// Example 1 - ConstantGap: ONE cam table, 9 points.
//
//   Mover 1 = master, runs at constant velocity around the track.
//   Mover 2 = slave, follows Mover 1 through a cam table that covers one full lap (1500 mm).
//
// Mover 2 is 100 mm behind Mover 1 on the straights and 60 mm in the curves, blended over TRANSITION mm
// at the start of every section. The table is written by hand in the action BuildTable (F_CamPoint).
//
// How to run (online view, with MAIN.eExample = ConstantGap):  bStart -> watch eState -> bStop.   On Error: bReset.
// Watch fGapActual while it runs: 100 on the straights, 60 in the curves, a smooth blend at each section start.
PROGRAM PRG_Example1
VAR CONSTANT
	// --- track geometry (mm) ---
	TRACK_LENGTH			: LREAL := 1500.0;	// = modulo factor of both mover axes
	STRAIGHT_1_START		: LREAL := 0.0;
	CURVE_1_START			: LREAL := 250.0;
	STRAIGHT_2_START		: LREAL := 750.0;
	CURVE_2_START			: LREAL := 1000.0;

	// --- wanted distance Mover 1 -> Mover 2 (mm, Mover 2 runs BEHIND Mover 1) ---
	GAP_STRAIGHT			: LREAL := 100.0;
	GAP_CURVE				: LREAL := 60.0;
	TRANSITION				: LREAL := 100.0;	// master travel over which the gap blends to the new value

	// --- demo dynamics ---
	MASTER_VELOCITY			: LREAL := 300.0;	// mm/s, Mover 1 while running
	POSITIONING_VELOCITY	: LREAL := 200.0;	// mm/s, Mover 2 while pre-positioning

	CAM_TABLE_ID			: MC_CAM_ID := 1;	// NC > Tables > Table 1 (Ex 1-4) > Mover 2
	CAM_POINTS				: UDINT := 9;
END_VAR
VAR
	// --- commands: set TRUE in the online view, they reset themselves ---
	bStart				: BOOL;
	bStop				: BOOL;
	bReset				: BOOL;
	eState				: E_State;

	// --- cam table data: CAM_POINTS points, loaded into NC table CAM_TABLE_ID ---
	aCamPoints			: ARRAY[1..CAM_POINTS] OF MC_MotionFunctionPoint;
	stCamTable			: MC_CAM_REF;

	// --- function blocks ---
	fbPowerMover1		: MC_Power;
	fbPowerMover2		: MC_Power;
	fbResetMover1		: MC_Reset;
	fbResetMover2		: MC_Reset;
	fbCamTableSelect	: MC_CamTableSelect;			// PLC array -> NC cam table
	fbReadTable			: MC_ReadCamTableSlaveDynamics;	// "where does the table want the slave for this master position?"
	fbMoveRelMover2		: MC_MoveRelative;
	fbCamIn				: MC_CamIn;
	fbMoveVeloMover1	: MC_MoveVelocity;
	fbHaltMover1		: MC_Halt;
	fbCamOut			: MC_CamOut;

	// --- live values worth watching ---
	fMover1Pos			: LREAL;	// modulo set position of Mover 1 (0..1500)
	fMover2Pos			: LREAL;	// modulo set position of Mover 2 (0..1500)
	fGapActual			: LREAL;	// how far Mover 2 is behind Mover 1 right now (along the track)
	fGapWanted			: LREAL;	// what the table asked for at coupling time
	bError				: BOOL;
	nErrorID			: UDINT;
END_VAR

// update axis status every cycle
GVL_Axes.Mover1();
GVL_Axes.Mover2();

// live gap: Mover 1 position minus Mover 2 position, wrapped to 0..1500
fMover1Pos := GVL_Axes.Mover1.NcToPlc.ModuloSetPos;
fMover2Pos := GVL_Axes.Mover2.NcToPlc.ModuloSetPos;
fGapActual := fMover1Pos - fMover2Pos;
IF fGapActual < 0.0 THEN
	fGapActual := fGapActual + TRACK_LENGTH;
END_IF

CASE eState OF
	E_State.Idle:
		IF bStart THEN
			bStart := FALSE;
			eState := E_State.Enable;
		END_IF

	E_State.Enable:
		fbPowerMover1.Enable := TRUE;
		fbPowerMover1.Enable_Positive := TRUE;
		fbPowerMover1.Enable_Negative := TRUE;
		fbPowerMover2.Enable := TRUE;
		fbPowerMover2.Enable_Positive := TRUE;
		fbPowerMover2.Enable_Negative := TRUE;
		IF fbPowerMover1.Status AND fbPowerMover2.Status THEN
			eState := E_State.Decouple;
		END_IF

	E_State.Decouple:
		// An earlier run may have left Mover 2 coupled: the NC keeps the coupling through an axis error and MC_Reset
		// does not clear it. MC_CamTableSelect refuses to overwrite a table that a coupled axis is using (0x4A26).
		IF NOT fbCamOut.Execute THEN
			IF GVL_Axes.Mover2.Status.Coupled THEN
				fbCamOut.Execute := TRUE;
			ELSE
				eState := E_State.BuildTable;
			END_IF
		ELSIF fbCamOut.Done THEN
			fbCamOut.Execute := FALSE;
			eState := E_State.BuildTable;
		END_IF

	E_State.BuildTable:
		// fill the point array once, then hand it to the NC (overwrites cam table CAM_TABLE_ID)
		IF NOT fbCamTableSelect.Execute THEN
			BuildTable();
		END_IF
		fbCamTableSelect.Periodic := TRUE;		// one table = one lap, repeat forever
		fbCamTableSelect.CamTableID := CAM_TABLE_ID;
		fbCamTableSelect.Execute := TRUE;
		IF fbCamTableSelect.Done THEN
			fbCamTableSelect.Execute := FALSE;
			eState := E_State.ReadTable;
		END_IF

	E_State.ReadTable:
		// Mover 1 stays where it is. Ask the NC what slave position the table wants for it.
		// The table master runs 0..1500 = the track, so Mover 1's track position goes in as it is.
		fbReadTable.CamTableID := CAM_TABLE_ID;
		fbReadTable.MasterPosition := fMover1Pos;
		fbReadTable.Execute := TRUE;
		IF fbReadTable.Done THEN
			fbReadTable.Execute := FALSE;
			// table: slave = master - gap   ->   gap = master - slave
			fGapWanted := fMover1Pos - fbReadTable.SlavePosition;
			// Mover 1 stands still, so this relative move can never run into it:
			// positive = Mover 2 closes up from behind, negative = Mover 2 backs off a little
			fbMoveRelMover2.Distance := fGapActual - fGapWanted;
			eState := E_State.Preposition;
		END_IF

	E_State.Preposition:
		fbMoveRelMover2.Velocity := POSITIONING_VELOCITY;
		fbMoveRelMover2.Execute := TRUE;
		IF fbMoveRelMover2.Done THEN
			fbMoveRelMover2.Execute := FALSE;
			eState := E_State.CamIn;
		END_IF

	E_State.CamIn:
		fbCamIn.CamTableID := CAM_TABLE_ID;
		fbCamIn.StartMode := MC_STARTMODE_ABSOLUTE;		// table master axis = Mover 1 track position
		fbCamIn.MasterOffset := 0.0;
		fbCamIn.SlaveOffset := 0.0;
		fbCamIn.MasterScaling := 1.0;
		fbCamIn.SlaveScaling := 1.0;
		// let the NC pick the slave offset so Mover 2 never jumps at coupling.
		// After the pre-positioning above that offset is 0 (or whole laps), so the table gaps apply 1:1.
		fbCamIn.Options.SlaveScalingMode := MC_CAMSCALING_AUTOOFFSET;
		fbCamIn.Execute := TRUE;
		IF fbCamIn.InSync THEN
			fbCamIn.Execute := FALSE;
			eState := E_State.Run;
		END_IF

	E_State.Run:
		// only the master is commanded - the slave is driven by the cam
		fbMoveVeloMover1.Velocity := MASTER_VELOCITY;
		fbMoveVeloMover1.Direction := MC_Positive_Direction;
		fbMoveVeloMover1.Execute := TRUE;
		IF bStop THEN
			bStop := FALSE;
			fbMoveVeloMover1.Execute := FALSE;
			eState := E_State.Stopping;
		END_IF

	E_State.Stopping:
		fbHaltMover1.Execute := TRUE;
		IF fbHaltMover1.Done THEN
			fbHaltMover1.Execute := FALSE;
			eState := E_State.CamOut;
		END_IF

	E_State.CamOut:
		fbCamOut.Execute := TRUE;
		IF fbCamOut.Done THEN
			fbCamOut.Execute := FALSE;
			eState := E_State.Idle;
		END_IF

	E_State.Error:
		fbCamTableSelect.Execute := FALSE;
		fbReadTable.Execute := FALSE;
		fbMoveRelMover2.Execute := FALSE;
		fbCamIn.Execute := FALSE;
		fbMoveVeloMover1.Execute := FALSE;
		// a slave error does not stop the master: halt Mover 1 if it is still running and not in error itself
		fbHaltMover1.Execute := NOT GVL_Axes.Mover1.Status.Error AND GVL_Axes.Mover1.Status.Moving;
		fbCamOut.Execute := FALSE;
		IF bReset THEN
			bReset := FALSE;
			fbResetMover1.Execute := TRUE;
			fbResetMover2.Execute := TRUE;
			eState := E_State.Resetting;
		END_IF

	E_State.Resetting:
		IF (fbResetMover1.Done OR fbResetMover1.Error) AND (fbResetMover2.Done OR fbResetMover2.Error) THEN
			fbResetMover1.Execute := FALSE;
			fbResetMover2.Execute := FALSE;
			bError := FALSE;
			nErrorID := 0;
			eState := E_State.Idle;
		END_IF
END_CASE

// any error anywhere -> Error state
IF eState <> E_State.Error AND eState <> E_State.Resetting THEN
	IF GVL_Axes.Mover1.Status.Error THEN
		nErrorID := GVL_Axes.Mover1.Status.ErrorID;
	ELSIF GVL_Axes.Mover2.Status.Error THEN
		nErrorID := GVL_Axes.Mover2.Status.ErrorID;
	ELSIF fbPowerMover1.Error THEN
		nErrorID := fbPowerMover1.ErrorID;
	ELSIF fbPowerMover2.Error THEN
		nErrorID := fbPowerMover2.ErrorID;
	ELSIF fbCamTableSelect.Error THEN
		nErrorID := fbCamTableSelect.ErrorID;
	ELSIF fbReadTable.Error THEN
		nErrorID := fbReadTable.ErrorID;
	ELSIF fbMoveRelMover2.Error THEN
		nErrorID := fbMoveRelMover2.ErrorID;
	ELSIF fbCamIn.Error THEN
		nErrorID := fbCamIn.ErrorID;
	ELSIF fbMoveVeloMover1.Error THEN
		nErrorID := fbMoveVeloMover1.ErrorID;
	ELSIF fbHaltMover1.Error THEN
		nErrorID := fbHaltMover1.ErrorID;
	ELSIF fbCamOut.Error THEN
		nErrorID := fbCamOut.ErrorID;
	END_IF
	IF nErrorID <> 0 THEN
		bError := TRUE;
		eState := E_State.Error;
	END_IF
END_IF

// call every function block once per cycle
fbPowerMover1(Axis := GVL_Axes.Mover1);
fbPowerMover2(Axis := GVL_Axes.Mover2);
fbResetMover1(Axis := GVL_Axes.Mover1);
fbResetMover2(Axis := GVL_Axes.Mover2);
fbCamTableSelect(Master := GVL_Axes.Mover1, Slave := GVL_Axes.Mover2, CamTable := stCamTable);
fbReadTable();
fbMoveRelMover2(Axis := GVL_Axes.Mover2);
fbCamIn(Master := GVL_Axes.Mover1, Slave := GVL_Axes.Mover2);
fbMoveVeloMover1(Axis := GVL_Axes.Mover1);
fbHaltMover1(Axis := GVL_Axes.Mover1);
fbCamOut(Slave := GVL_Axes.Mover2);

ACTION BuildTable:
// One lap of Mover 1 (0..1500) -> where Mover 2 has to be (master minus gap).
// Every section starts with a TRANSITION where the gap blends to the new value, then runs 1:1.
// The curve type on a point is used from that point to the NEXT point.
//
//                          idx  master position                gap           curve to next point
aCamPoints[1] := F_CamPoint(1,   STRAIGHT_1_START,              GAP_CURVE,    MOTIONFUNCTYPE_POLYNOM5_MM);	//    0: still 60 from the curve before, blend to 100
aCamPoints[2] := F_CamPoint(2,   STRAIGHT_1_START + TRANSITION, GAP_STRAIGHT, MOTIONFUNCTYPE_POLYNOM1);		//  100: 1:1, 100 behind
aCamPoints[3] := F_CamPoint(3,   CURVE_1_START,                 GAP_STRAIGHT, MOTIONFUNCTYPE_POLYNOM5_MM);	//  250: blend to 60
aCamPoints[4] := F_CamPoint(4,   CURVE_1_START + TRANSITION,    GAP_CURVE,    MOTIONFUNCTYPE_POLYNOM1);		//  350: 1:1, 60 behind
aCamPoints[5] := F_CamPoint(5,   STRAIGHT_2_START,              GAP_CURVE,    MOTIONFUNCTYPE_POLYNOM5_MM);	//  750: blend to 100
aCamPoints[6] := F_CamPoint(6,   STRAIGHT_2_START + TRANSITION, GAP_STRAIGHT, MOTIONFUNCTYPE_POLYNOM1);		//  850: 1:1, 100 behind
aCamPoints[7] := F_CamPoint(7,   CURVE_2_START,                 GAP_STRAIGHT, MOTIONFUNCTYPE_POLYNOM5_MM);	// 1000: blend to 60
aCamPoints[8] := F_CamPoint(8,   CURVE_2_START + TRANSITION,    GAP_CURVE,    MOTIONFUNCTYPE_POLYNOM1);		// 1100: 1:1, 60 behind
aCamPoints[9] := F_CamPoint(9,   TRACK_LENGTH,                  GAP_CURVE,    MOTIONFUNCTYPE_POLYNOM1);		// 1500: end of lap, same gap as point 1
aCamPoints[9].RelIndexNextPoint := 0;	// last point has no successor

// Slave goes from -60 (point 1) to 1440 (point 9) = +1500 per lap. The NC calls this a "cyclic cam
// with lift" and simply keeps adding 1500 every lap, so Mover 2 keeps going around with Mover 1.

// describe the array to the NC
stCamTable.pArray		:= ADR(aCamPoints);
stCamTable.ArraySize	:= SIZEOF(aCamPoints);
stCamTable.TableType	:= MC_TABLETYPE_MOTIONFUNCTION;
stCamTable.NoOfRows		:= CAM_POINTS;
stCamTable.NoOfColumns	:= 1;
END_ACTION

END_PROGRAM

(* stored: Version 1.1.0.1
   POU PRG_Example1: Id {5e36387e-9ed2-439e-b8e3-3c803a97c1ff}, SpecialFunc None
   Action BuildTable: Id {4f47832a-288c-4251-ac75-f5a613e177ab} *)
